{attribute 'linkalways'} 
{attribute 'no_explicit_call' := 'This FB is a CLASS and must be accessed using methods or properties'}
{attribute 'enable_dynamic_creation'}
FUNCTION_BLOCK SessionManager implements I_SessionManager, I_SessionStorage
VAR
	activeSessions : Dictionary;
	sessionIdGenerator : I_SessionIdGenerator;
	currentStorageId : UDINT;
	sessionMaxLife : TIME;
END_VAR

METHOD PUBLIC CheckForExpiredSessions
VAR_INPUT
END_VAR
VAR
	enumerator : I_ForwardEnumerator;
	session : I_Session;
	expiredSessions : Stack;
END_VAR
enumerator := activeSessions.GetEnumerator();

WHILE enumerator.MoveNext() DO
	IF enumerator.TryGet(session) THEN
		IF session.LastAccessedTimestamp.IsDurationElapsed(sessionMaxLife) THEN
			expiredSessions.Push(session);
		END_IF
	END_IF
END_WHILE

enumerator.Dispose();

WHILE expiredSessions.TryPop(session) DO
	DisposeSession(session.Id);
END_WHILE
END_METHOD

METHOD PRIVATE CreateNewSession : I_Session
VAR
	id : T_MAXSTRING;
	pSession : POINTER TO Session;
END_VAR
id := sessionIdGenerator.Generate();
pSession := __NEW(Session(SessionId := id));
CreateNewSession := pSession^;
END_METHOD

METHOD PUBLIC CreateSession : T_MAXSTRING;
VAR
	session : I_Session;
END_VAR
session := CreateNewSession();
activeSessions.AddOrUpdate(session.Id, session);
CreateSession := session.Id;
END_METHOD

METHOD PUBLIC CyclicCall
VAR_INPUT
END_VAR
CheckForExpiredSessions();
END_METHOD

METHOD PUBLIC DisposeAllSessions
VAR_INPUT
END_VAR
VAR
	enumerator : I_ForwardEnumerator;
	session : I_Session;
END_VAR
enumerator := activeSessions.GetEnumerator();

WHILE enumerator.MoveNext() DO
	if enumerator.TryGet(session) then
		session.Dispose();
	END_IF
END_WHILE

enumerator.Dispose();
activeSessions.Clear();
END_METHOD

METHOD PUBLIC DisposeSession
VAR_INPUT
	Id : T_MAXSTRING;
END_VAR
VAR
	session : I_Session;
END_VAR
IF NOT activeSessions.TryGetValue(Id, session) THEN
	RETURN;
END_IF

session.Dispose();
activeSessions.Remove(Id);
END_METHOD

METHOD PUBLIC DisposeSessionDataById
VAR_INPUT
	SessionId : T_MAXSTRING;
	StorageId : T_MAXSTRING;
END_VAR
VAR
	session : I_Session;
	sessionData : I_SessionData;
END_VAR
IF StorageId = '' THEN 
	RETURN;
END_IF

IF NOT activeSessions.TryGetValue(SessionId, session) THEN
	RETURN;
END_IF

IF NOT session.TryGetDataFromStorage(StorageId, sessionData) THEN
	RETURN;
END_IF

session.DisposeDataFromStorage(StorageId);
END_METHOD

METHOD FB_exit : BOOL
VAR_INPUT
	bInCopyCode : BOOL; // if TRUE, the exit method is called for exiting an instance that is copied afterwards (online change).
END_VAR
IF bInCopyCode THEN
	RETURN;
END_IF

DisposeAllSessions();
END_METHOD

METHOD FB_init : BOOL
VAR_INPUT
	bInitRetains : BOOL; // if TRUE, the retain variables are initialized (warm start / cold start)
	bInCopyCode : BOOL;  // if TRUE, the instance afterwards gets moved into the copy code (online change)
	SessionIdGenerator : I_SessionIdGenerator;
	SessionMaxLife : TIME;
END_VAR
THIS^.sessionIdGenerator := SessionIdGenerator;
THIS^.sessionMaxLife := SessionMaxLife;
END_METHOD

METHOD PUBLIC IsValidSession : BOOL
VAR_INPUT
	Id : T_MAXSTRING;
END_VAR
IsValidSession := activeSessions.ContainsKey(Id);
END_METHOD

PROPERTY PUBLIC SessionCount : DINT
GET
SessionCount := activeSessions.Count;
END_GET
END_PROPERTY

METHOD PUBLIC TryRetreiveSessionDataById : BOOL
VAR_INPUT
	SessionId : T_MAXSTRING;
	StorageId : T_MAXSTRING;
	Destination : REFERENCE TO I_SessionData;
END_VAR
VAR
	session : I_Session;
END_VAR
IF NOT activeSessions.TryGetValue(SessionId, session) THEN
	RETURN;
END_IF

TryRetreiveSessionDataById := session.TryGetDataFromStorage(StorageId, Destination);
END_METHOD

METHOD PUBLIC TryStoreSessionDataById : BOOL
VAR_INPUT
	SessionId : T_MAXSTRING;
	StorageId : T_MAXSTRING;
	Source : I_SessionData;
END_VAR
VAR
	session : I_Session;
END_VAR
IF StorageId = '' THEN 
	RETURN;
END_IF

IF NOT activeSessions.TryGetValue(SessionId, session) THEN
	RETURN;
END_IF

session.AddOrUpdateStorage(StorageId, Source);
TryStoreSessionDataById := TRUE;
END_METHOD

END_FUNCTION_BLOCK

(* stored: Version 1.1.0.1, ProductVersion 3.1.4024.12
   POU SessionManager: Id {90fd976c-1ca7-4040-ad52-5f45d1d6b3c4}, SpecialFunc None
   Folder Constructor: Id {7dc71ecd-1e2e-4054-be7b-88439bd7a055}
   Folder Destructor: Id {955b78d7-748c-465a-8ef1-8ade3a09e309}
   Folder Private: Id {0e592bc1-44ed-4d2b-bc39-bf9cda67de39}
   Method CheckForExpiredSessions: Id {ed802867-966f-4b09-bf99-0d8bc76df646}
   Method CreateNewSession: Id {8f73492b-d285-4067-945e-51553f07c17c}
   Method CreateSession: Id {ae54ac8f-e99b-4edc-a710-65a4bc03a4b0}
   Method CyclicCall: Id {adca83ea-788a-4205-a0b0-cc70c54d65e7}
   Method DisposeAllSessions: Id {b0328bcc-a2a7-45fb-bb30-b127df358c87}
   Method DisposeSession: Id {1f8b0e18-85fa-48f8-b1fa-f14505dc3153}
   Method DisposeSessionDataById: Id {1ad28fbf-1f29-4da3-a785-67b66326e540}
   Method FB_exit: Id {43f8357b-dbc8-4eff-8238-652c04179c2b}
   Method FB_init: Id {fe268b30-f722-40e5-921d-eba5791b3d9f}
   Method IsValidSession: Id {31c4bdcd-d6c8-444d-8b15-ff5226cc4a5a}
   Property SessionCount: Id {3649ded8-410b-44c9-babc-17c1bc3784d7}
   Get Get: Id {a30c1e41-1077-4bd5-b1bb-dbf3345d9355}
   Method TryRetreiveSessionDataById: Id {0fb427b1-5ae2-4f38-94c9-bdd72a673e66}
   Method TryStoreSessionDataById: Id {23603274-63a2-4b38-b5eb-0241b0d13401} *)
